VAR_GLOBAL
	stBPTime			:	ST_PumpTime;
	stIntHeatCirTime	:	ST_PumpTime;
	nMaxPre				:	DWORD;
END_VAR

(* stored: Version 1.1.0.1, ProductVersion 3.1.4018.2
   GVL PumpTiming: Id {829ac6aa-6c7c-4148-8eca-ed010515632e} *)
